// TIA Portal V19 export
TYPE "LEXCHANGETRAY_typeVfdContronNodeMonitoring"
// simulated: Bool
// vfdStopped: Bool
// monitoring: LBC_typeSinaSpeedControlNodeMonitoring
// stored: Access Published
   STRUCT
      simulated : Bool;
      vfdStopped : Bool;
      monitoring : "LBC_typeSinaSpeedControlNodeMonitoring";
   END_STRUCT;
END_TYPE
